REGION Network 90: SALIDAS - Girar a 0º
   RUNG wire#powerrail
      Contact( #Selec_M1_Entrada )
      wire#w1
      I_Contact( #PosMG_0 )
      I_Contact( #STAT_MGRetroBuscarPos )
      wire#w2
      Contact( #EstadoZona.Marcha_CBx )
      I_Contact( #EstadoVI.Error_Mx )
      I_Contact( #Error_Tx )
      Coil( #MA_Giro_0 )
   END_RUNG
   RUNG wire#powerrail
      Contact( #Selec_M1_Salida )
      Contact( #SaliendoCarga )
   END_RUNG wire#w1
   RUNG wire#powerrail
      Contact( #Selec_M3_Entrada )
   END_RUNG wire#w1
   RUNG wire#powerrail
      Contact( #Selec_M3_Salida )
      Contact( #SaliendoCarga )
   END_RUNG wire#w1
   RUNG wire#powerrail
      Contact( #PosMG_EnReposo_0 )
      Contact( #Mx_ET01 )
   END_RUNG wire#w1
   RUNG wire#powerrail
      Contact( #Selec_M2_Entrada )
      wire#w3
      I_Contact( #PosMG_90 )
      Contact( #STAT_MGRetroBuscarPos )
   END_RUNG wire#w2
   RUNG wire#powerrail
      Contact( #Selec_M2_Salida )
      Contact( #SaliendoCarga )
   END_RUNG wire#w3
   RUNG wire#powerrail
      Contact( #Selec_M4_Entrada )
   END_RUNG wire#w3
   RUNG wire#powerrail
      Contact( #Selec_M4_Salida )
      Contact( #SaliendoCarga )
   END_RUNG wire#w3
   RUNG wire#powerrail
      Contact( #PosMG_EnReposo_90 )
      Contact( #Mx_ET01 )
   END_RUNG wire#w3
   // the same network as SCL:
   #MA_Giro_0 := (((#Selec_M1_Entrada OR (#Selec_M1_Salida AND #SaliendoCarga) OR #Selec_M3_Entrada OR (#Selec_M3_Salida AND #SaliendoCarga) OR (#PosMG_EnReposo_0 AND #Mx_ET01)) AND NOT #PosMG_0 AND NOT #STAT_MGRetroBuscarPos) OR ((#Selec_M2_Entrada OR (#Selec_M2_Salida AND #SaliendoCarga) OR #Selec_M4_Entrada OR (#Selec_M4_Salida AND #SaliendoCarga) OR (#PosMG_EnReposo_90 AND #Mx_ET01)) AND NOT #PosMG_90 AND #STAT_MGRetroBuscarPos)) AND #EstadoZona.Marcha_CBx AND NOT #EstadoVI.Error_Mx AND NOT #Error_Tx;
END_REGION

REGION Network 91: SALIDAS - Girar a 90º
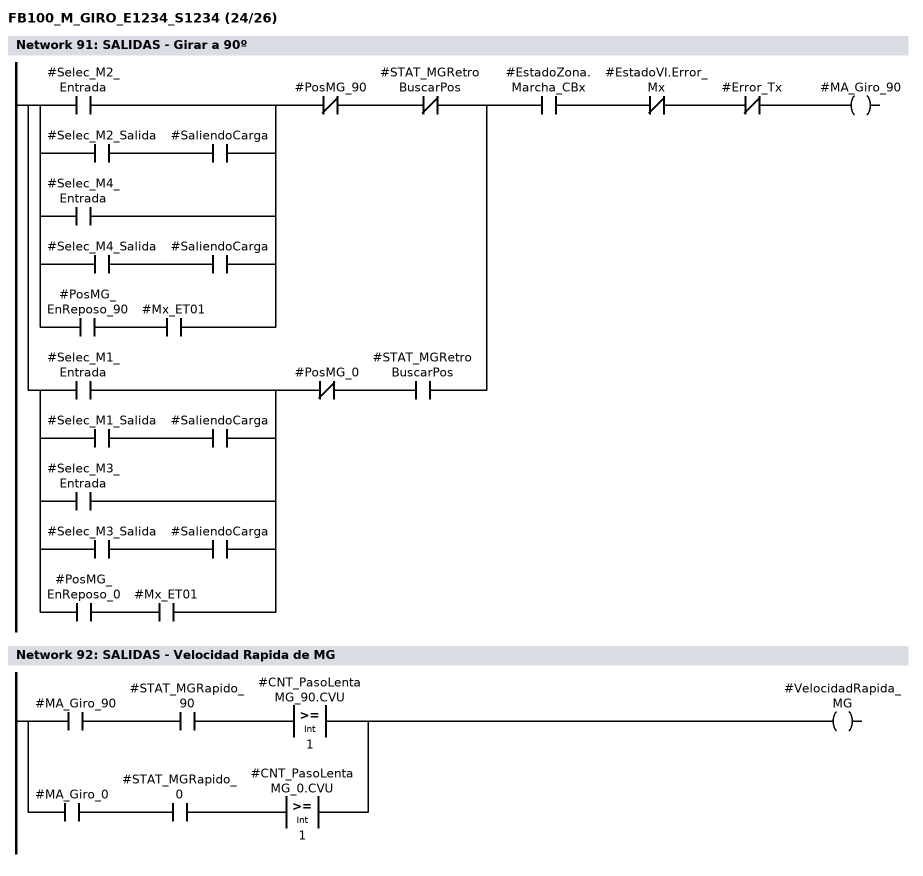
   RUNG wire#powerrail
      Contact( #Selec_M2_Entrada )
      wire#w1
      I_Contact( #PosMG_90 )
      I_Contact( #STAT_MGRetroBuscarPos )
      wire#w2
      Contact( #EstadoZona.Marcha_CBx )
      I_Contact( #EstadoVI.Error_Mx )
      I_Contact( #Error_Tx )
      Coil( #MA_Giro_90 )
   END_RUNG
   RUNG wire#powerrail
      Contact( #Selec_M2_Salida )
      Contact( #SaliendoCarga )
   END_RUNG wire#w1
   RUNG wire#powerrail
      Contact( #Selec_M4_Entrada )
   END_RUNG wire#w1
   RUNG wire#powerrail
      Contact( #Selec_M4_Salida )
      Contact( #SaliendoCarga )
   END_RUNG wire#w1
   RUNG wire#powerrail
      Contact( #PosMG_EnReposo_90 )
      Contact( #Mx_ET01 )
   END_RUNG wire#w1
   RUNG wire#powerrail
      Contact( #Selec_M1_Entrada )
      wire#w3
      I_Contact( #PosMG_0 )
      Contact( #STAT_MGRetroBuscarPos )
   END_RUNG wire#w2
   RUNG wire#powerrail
      Contact( #Selec_M1_Salida )
      Contact( #SaliendoCarga )
   END_RUNG wire#w3
   RUNG wire#powerrail
      Contact( #Selec_M3_Entrada )
   END_RUNG wire#w3
   RUNG wire#powerrail
      Contact( #Selec_M3_Salida )
      Contact( #SaliendoCarga )
   END_RUNG wire#w3
   RUNG wire#powerrail
      Contact( #PosMG_EnReposo_0 )
      Contact( #Mx_ET01 )
   END_RUNG wire#w3
   // the same network as SCL:
   #MA_Giro_90 := (((#Selec_M2_Entrada OR (#Selec_M2_Salida AND #SaliendoCarga) OR #Selec_M4_Entrada OR (#Selec_M4_Salida AND #SaliendoCarga) OR (#PosMG_EnReposo_90 AND #Mx_ET01)) AND NOT #PosMG_90 AND NOT #STAT_MGRetroBuscarPos) OR ((#Selec_M1_Entrada OR (#Selec_M1_Salida AND #SaliendoCarga) OR #Selec_M3_Entrada OR (#Selec_M3_Salida AND #SaliendoCarga) OR (#PosMG_EnReposo_0 AND #Mx_ET01)) AND NOT #PosMG_0 AND #STAT_MGRetroBuscarPos)) AND #EstadoZona.Marcha_CBx AND NOT #EstadoVI.Error_Mx AND NOT #Error_Tx;
END_REGION

REGION Network 92: SALIDAS - Velocidad Rapida de MG
   RUNG wire#powerrail
      Contact( #MA_Giro_90 )
      Contact( #STAT_MGRapido_90 )
      { S7_Templates := "SrcType := Int" } GE_Contact(in1 := #CNT_PasoLentaMG_90.CVU, in2 := 1)
      wire#w1
      Coil( #VelocidadRapida_MG )
   END_RUNG
   RUNG wire#powerrail
      Contact( #MA_Giro_0 )
      Contact( #STAT_MGRapido_0 )
      { S7_Templates := "SrcType := Int" } GE_Contact(in1 := #CNT_PasoLentaMG_0.CVU, in2 := 1)
   END_RUNG wire#w1
   // the same network as SCL:
   #VelocidadRapida_MG := (#MA_Giro_90 AND #STAT_MGRapido_90 AND (#CNT_PasoLentaMG_90.CVU >= 1)) OR (#MA_Giro_0 AND #STAT_MGRapido_0 AND (#CNT_PasoLentaMG_0.CVU >= 1));
END_REGION

REGION Network 93: ESTADOS DE LA MESA
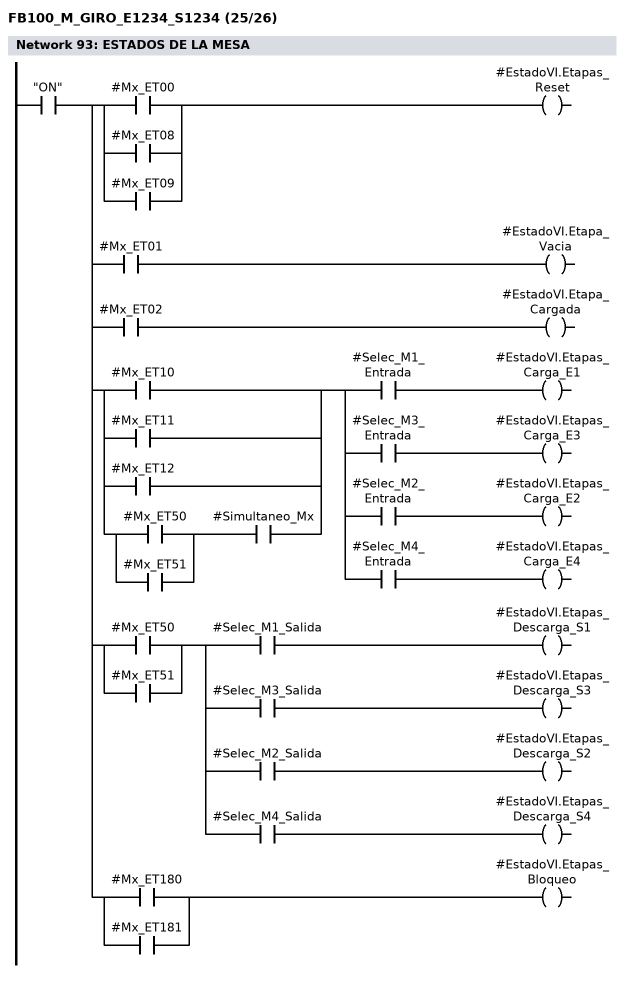
   RUNG wire#powerrail
      Contact( "ON" )
      wire#w1
      Contact( #Mx_ET00 )
      wire#w2
      Coil( #EstadoVI.Etapas_Reset )
   END_RUNG
   RUNG wire#w1
      Contact( #Mx_ET08 )
   END_RUNG wire#w2
   RUNG wire#w1
      Contact( #Mx_ET09 )
   END_RUNG wire#w2
   RUNG wire#w1
      Contact( #Mx_ET01 )
      Coil( #EstadoVI.Etapa_Vacia )
   END_RUNG
   RUNG wire#w1
      Contact( #Mx_ET02 )
      Coil( #EstadoVI.Etapa_Cargada )
   END_RUNG
   RUNG wire#w1
      Contact( #Mx_ET10 )
      wire#w3
      Contact( #Selec_M1_Entrada )
      Coil( #EstadoVI.Etapas_Carga_E1 )
   END_RUNG
   RUNG wire#w1
      Contact( #Mx_ET11 )
   END_RUNG wire#w3
   RUNG wire#w1
      Contact( #Mx_ET12 )
   END_RUNG wire#w3
   RUNG wire#w1
      Contact( #Mx_ET50 )
      wire#w4
      Contact( #Simultaneo_Mx )
   END_RUNG wire#w3
   RUNG wire#w1
      Contact( #Mx_ET51 )
   END_RUNG wire#w4
   RUNG wire#w3
      Contact( #Selec_M3_Entrada )
      Coil( #EstadoVI.Etapas_Carga_E3 )
   END_RUNG
   RUNG wire#w3
      Contact( #Selec_M2_Entrada )
      Coil( #EstadoVI.Etapas_Carga_E2 )
   END_RUNG
   RUNG wire#w3
      Contact( #Selec_M4_Entrada )
      Coil( #EstadoVI.Etapas_Carga_E4 )
   END_RUNG
   RUNG wire#w1
      Contact( #Mx_ET50 )
      wire#w5
      Contact( #Selec_M1_Salida )
      Coil( #EstadoVI.Etapas_Descarga_S1 )
   END_RUNG
   RUNG wire#w1
      Contact( #Mx_ET51 )
   END_RUNG wire#w5
   RUNG wire#w5
      Contact( #Selec_M3_Salida )
      Coil( #EstadoVI.Etapas_Descarga_S3 )
   END_RUNG
   RUNG wire#w5
      Contact( #Selec_M2_Salida )
      Coil( #EstadoVI.Etapas_Descarga_S2 )
   END_RUNG
   RUNG wire#w5
      Contact( #Selec_M4_Salida )
      Coil( #EstadoVI.Etapas_Descarga_S4 )
   END_RUNG
   RUNG wire#w1
      Contact( #Mx_ET180 )
      wire#w6
      Coil( #EstadoVI.Etapas_Bloqueo )
   END_RUNG
   RUNG wire#w1
      Contact( #Mx_ET181 )
   END_RUNG wire#w6
   // the same network as SCL:
   #EstadoVI.Etapas_Reset := "ON" AND (#Mx_ET00 OR #Mx_ET08 OR #Mx_ET09);
   #EstadoVI.Etapa_Vacia := "ON" AND #Mx_ET01;
   #EstadoVI.Etapa_Cargada := "ON" AND #Mx_ET02;
   #_w1 := "ON" AND (#Mx_ET10 OR #Mx_ET11 OR #Mx_ET12 OR ((#Mx_ET50 OR #Mx_ET51) AND #Simultaneo_Mx));
   #EstadoVI.Etapas_Carga_E1 := #_w1 AND #Selec_M1_Entrada;
   #EstadoVI.Etapas_Carga_E3 := #_w1 AND #Selec_M3_Entrada;
   #EstadoVI.Etapas_Carga_E2 := #_w1 AND #Selec_M2_Entrada;
   #EstadoVI.Etapas_Carga_E4 := #_w1 AND #Selec_M4_Entrada;
   #_w2 := "ON" AND (#Mx_ET50 OR #Mx_ET51);
   #EstadoVI.Etapas_Descarga_S1 := #_w2 AND #Selec_M1_Salida;
   #EstadoVI.Etapas_Descarga_S3 := #_w2 AND #Selec_M3_Salida;
   #EstadoVI.Etapas_Descarga_S2 := #_w2 AND #Selec_M2_Salida;
   #EstadoVI.Etapas_Descarga_S4 := #_w2 AND #Selec_M4_Salida;
   #EstadoVI.Etapas_Bloqueo := "ON" AND (#Mx_ET180 OR #Mx_ET181);
END_REGION

REGION Network 94: ENTRADAS DE LA MESA
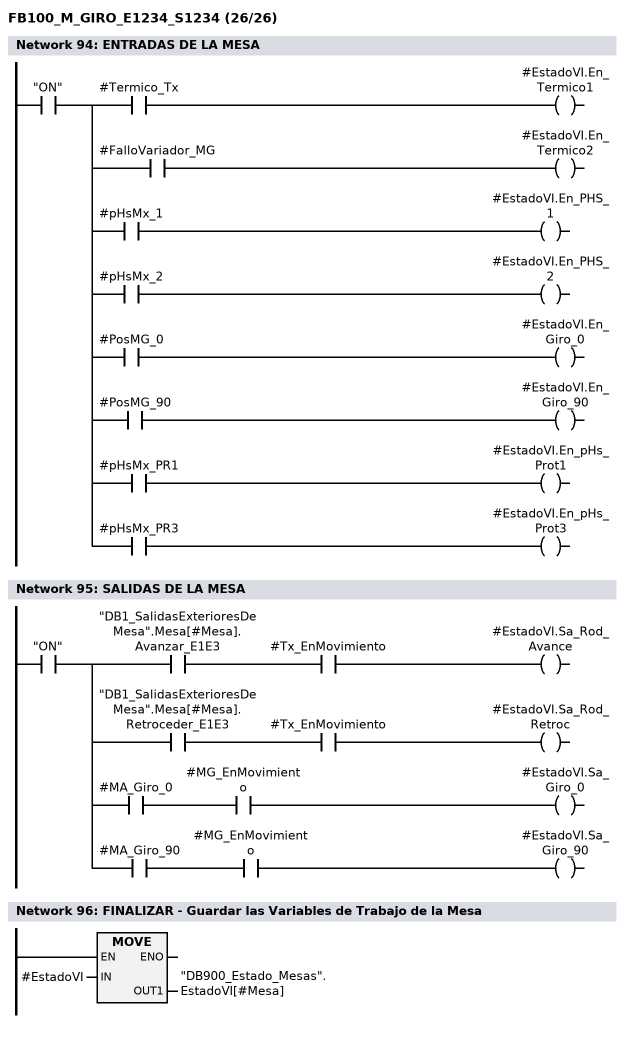
   RUNG wire#powerrail
      Contact( "ON" )
      wire#w1
      Contact( #Termico_Tx )
      Coil( #EstadoVI.En_Termico1 )
   END_RUNG
   RUNG wire#w1
      Contact( #FalloVariador_MG )
      Coil( #EstadoVI.En_Termico2 )
   END_RUNG
   RUNG wire#w1
      Contact( #pHsMx_1 )
      Coil( #EstadoVI.En_PHS_1 )
   END_RUNG
   RUNG wire#w1
      Contact( #pHsMx_2 )
      Coil( #EstadoVI.En_PHS_2 )
   END_RUNG
   RUNG wire#w1
      Contact( #PosMG_0 )
      Coil( #EstadoVI.En_Giro_0 )
   END_RUNG
   RUNG wire#w1
      Contact( #PosMG_90 )
      Coil( #EstadoVI.En_Giro_90 )
   END_RUNG
   RUNG wire#w1
      Contact( #pHsMx_PR1 )
      Coil( #EstadoVI.En_pHs_Prot1 )
   END_RUNG
   RUNG wire#w1
      Contact( #pHsMx_PR3 )
      Coil( #EstadoVI.En_pHs_Prot3 )
   END_RUNG
   // the same network as SCL:
   #EstadoVI.En_Termico1 := "ON" AND #Termico_Tx;
   #EstadoVI.En_Termico2 := "ON" AND #FalloVariador_MG;
   #EstadoVI.En_PHS_1 := "ON" AND #pHsMx_1;
   #EstadoVI.En_PHS_2 := "ON" AND #pHsMx_2;
   #EstadoVI.En_Giro_0 := "ON" AND #PosMG_0;
   #EstadoVI.En_Giro_90 := "ON" AND #PosMG_90;
   #EstadoVI.En_pHs_Prot1 := "ON" AND #pHsMx_PR1;
   #EstadoVI.En_pHs_Prot3 := "ON" AND #pHsMx_PR3;
END_REGION

REGION Network 95: SALIDAS DE LA MESA
   RUNG wire#powerrail
      Contact( "ON" )
      wire#w1
      Contact( "DB1_SalidasExterioresDeMesa".Mesa[#Mesa].Avanzar_E1E3 )
      Contact( #Tx_EnMovimiento )
      Coil( #EstadoVI.Sa_Rod_Avance )
   END_RUNG
   RUNG wire#w1
      Contact( "DB1_SalidasExterioresDeMesa".Mesa[#Mesa].Retroceder_E1E3 )
      Contact( #Tx_EnMovimiento )
      Coil( #EstadoVI.Sa_Rod_Retroc )
   END_RUNG
   RUNG wire#w1
      Contact( #MA_Giro_0 )
      Contact( #MG_EnMovimiento )
      Coil( #EstadoVI.Sa_Giro_0 )
   END_RUNG
   RUNG wire#w1
      Contact( #MA_Giro_90 )
      Contact( #MG_EnMovimiento )
      Coil( #EstadoVI.Sa_Giro_90 )
   END_RUNG
   // the same network as SCL:
   #EstadoVI.Sa_Rod_Avance := "ON" AND "DB1_SalidasExterioresDeMesa".Mesa[#Mesa].Avanzar_E1E3 AND #Tx_EnMovimiento;
   #EstadoVI.Sa_Rod_Retroc := "ON" AND "DB1_SalidasExterioresDeMesa".Mesa[#Mesa].Retroceder_E1E3 AND #Tx_EnMovimiento;
   #EstadoVI.Sa_Giro_0 := "ON" AND #MA_Giro_0 AND #MG_EnMovimiento;
   #EstadoVI.Sa_Giro_90 := "ON" AND #MA_Giro_90 AND #MG_EnMovimiento;
END_REGION

REGION Network 96: FINALIZAR - Guardar las Variables de Trabajo de la Mesa
   RUNG wire#powerrail
      Move(in := #EstadoVI, out1 => "DB900_Estado_Mesas".EstadoVI[#Mesa])
   END_RUNG
   // the same network as SCL:
   "DB900_Estado_Mesas".EstadoVI[#Mesa] := #EstadoVI;
END_REGION
END_FUNCTION_BLOCK
